FUNCTION_BLOCK StopMovementsAndProgramTask EXTENDS TcoAbbRoboticsTask
VAR

	_stopType: TcoAbstractions.eTcoRoboticsStopType;
END_VAR



IF Execute() THEN
	IF _progress = 0 THEN
		IF NOT __ISVALIDREF(inoControl) THEN
			_varInfo :=__VARINFO(inoControl);
			Messenger.Programming(_sb.Clear().Append('<#Invalid reference: #>').Append(_varInfo.Symbol).ToString()).Pin();
		ELSIF NOT __ISVALIDREF(inoConfig) THEN                                                  
			_varInfo :=__VARINFO(inoConfig);                                                    
			Messenger.Programming(_sb.Clear().Append('<#Invalid reference: #>').Append(_varInfo.Symbol).ToString()).Pin();
		ELSIF NOT __ISVALIDREF(inoStatus) THEN                                                  
			_varInfo :=__VARINFO(inoStatus);                                                    
			Messenger.Programming(_sb.Clear().Append('<#Invalid reference: #>').Append(_varInfo.Symbol).ToString()).Pin();
			ELSE
			_progress := _progress + 1;
		END_IF

	END_IF
	IF _progress = 1 THEN
		inoControl.SoftStop := TRUE;
		inoControl.QuickStop := FALSE;
	
		IF _stopType = TcoAbstractions.eTcoRoboticsStopType.Quick THEN
			inoControl.SoftStop := FALSE;
			inoControl.QuickStop := TRUE;
		END_IF
	
	
		IF inoStatus.State.MoveInactive THEN
			_progress := _progress + 1;
		END_IF
	END_IF;		

	IF _progress = 2 THEN
		inoControl.StopProgram:=TRUE;
		IF NOT inoStatus.State.CycleOn THEN
			_progress := _progress + 1;
		END_IF
	END_IF;		
	
	IF _progress = 3 THEN	
		inoControl.SoftStop := FALSE;
		inoControl.QuickStop := FALSE;
		inoControl.StopProgram:=FALSE;
	END_IF;		
		

    DoneWhen( inoStatus.State.MoveInactive AND NOT inoStatus.State.CycleOn);
    CallTimers(TRUE);
	
	THIS^.ThrowWhen(_errorTimer.Q);
END_IF

IF  THIS^.Error AND NOT _errorMessage.Pinned THEN
	THIS^.Restore();
END_IF

METHOD PUBLIC FB_init : BOOL
VAR_INPUT
    bInitRetains : BOOL; // if TRUE, the retain variables are initialized (warm start / cold start)
    bInCopyCode : BOOL; // if TRUE, the instance afterwards gets moved into the copy code (online change)
  	ParentObject : ITcoObject;	
END_VAR
END_METHOD

METHOD INTERNAL InvokeWithParams : ITcoTaskStatus
VAR_INPUT
	inStopType : eTcoRoboticsStopType;
END_VAR
_stopType := inStopType;
InvokeWithParams := THIS^.Invoke();
END_METHOD

(*~
	<docu>
		<summary>
			Executes when task is aborted.
		</summary>			
	</docu>	
~*)
METHOD PROTECTED OnAbort
IF  __ISVALIDREF(inoStatus) THEN   THIS^.inoStatus.ActionDescription := '<#Stop movements and program was aborted, while not yet completed!#>';END_IF; 
inoControl.SoftStop := FALSE;
inoControl.QuickStop := FALSE;
inoControl.StopProgram:=FALSE;
END_METHOD

(*~
	<docu>
		<summary>
			Executes when task reaches the ```Done``` state .
		</summary>			
	</docu>	
~*)
METHOD PROTECTED OnDone
IF  __ISVALIDREF(inoStatus) THEN  THIS^.inoStatus.ActionDescription := '<#Stop movements and program  was completed successfully.#>';END_IF; 
_progress:=0;
END_METHOD

(*~
	<docu>
		<summary>
			Executes when task reaches the ```Error``` state.
			
		</summary>			
	</docu>	
~*)
METHOD PROTECTED OnError
VAR
	description: STRING;
END_VAR
THIS^.inoStatus.ActionDescription := '<#Stop movements and program finished with error.#>';
IF  __ISVALIDREF(inoStatus) THEN   THIS^.inoStatus.ActionDescription := description; END_IF;
THIS^._errorMessage.Error(_sb.Clear().Append(description).Append(' To restore acknowledge this alarm.').ToString()).Pin();
END_METHOD

METHOD PROTECTED OnStart
IF  __ISVALIDREF(inoStatus) THEN  THIS^.inoStatus.ActionDescription := '<#Stop movements and program started.#>'; END_IF; 
CallTimers(FALSE);
END_METHOD

(*~
	<docu>
		<summary>
			Restores this instance to the Ready state. Can be called explicitly or from within one of the restore mechanisms.
			<para>
				See also <see cref="PlcDocu.TcoCore.TcoTask.AutoRestorable()"/>
			</para>
		</summary>			
	</docu>	
~*)
METHOD Restore : ITcoRestorable
SUPER^.Restore();
inoControl.SoftStop := FALSE;
inoControl.QuickStop := FALSE;
inoControl.StopProgram:=FALSE;
END_METHOD

END_FUNCTION_BLOCK

(* stored: Version 1.1.0.1, ProductVersion 3.1.4024.12
   POU StopMovementsAndProgramTask: Id {bbc19dcc-9bcd-0b3f-09de-7073c12da196}, SpecialFunc None
   Method FB_init: Id {fe08e306-c22d-0e6b-3c13-63ab1d6fa1bb}
   Method InvokeWithParams: Id {94750881-5ca5-0421-012f-835b9aa7a2b0}
   Method OnAbort: Id {6e6849be-c1e2-0cb8-00f0-d18e388fb8f8}
   Method OnDone: Id {51a8987e-1e66-08ef-1570-d67484cf25a2}
   Method OnError: Id {22f3ae59-de11-0e7f-2631-bb6d0b4b63fd}
   Method OnStart: Id {23130bcb-8225-07f0-048a-2722a360db86}
   Method Restore: Id {f6e004b9-78ef-0f57-24a2-3a86a8d50611} *)
